// TIA Portal V17 export
// export: Created 2023-10-18T08:31:00.1217102Z, ExportSetting WithDefaults, WithReadOnly, DisplayName Totally Integrated Automation Portal, DisplayVersion V16 Update 4, DisplayName TIA Portal Version Control Interface, DisplayVersion V16 Update 2, DisplayName TIA Portal Openness, DisplayVersion V16 Update 4, DisplayName SINAMICS Startdrive Advanced, DisplayVersion V16 Update 5, DisplayName SINAMICS Startdrive G130, G150, S120, S150, SINAMICS MV, S210, DisplayVersion V16 Update 5, DisplayName SINAMICS Startdrive G110M, G120, G120C, G120D, G120P, G115D, DisplayVersion V16 Update 5, DisplayName STEP 7 Professional, DisplayVersion V16 Update 4, DisplayName STEP 7 Safety, DisplayVersion V16, DisplayName SINUMERIK 840D sl STEP 7 Toolbox, DisplayVersion V16 Update 2, DisplayName WinCC Advanced, DisplayVersion V16 Update 4
FUNCTION "AF_Safety" : Void   // FC2, FBD
{ S7_Optimized_Access := 'TRUE' }
VERSION : 0.1
// stored: AutoNumber true, CodeModifiedDate 2023-08-03T13:12:21.5628456Z, CompileDate 2023-08-03T13:12:26.4065718Z, CreationDate 2023-06-02T14:39:29.8490668Z, HandleErrorsWithinBlock false, InterfaceModifiedDate 2023-06-02T14:39:29.8490668Z, IsConsistent true, IsIECCheckEnabled false, IsKnowHowProtected false, IsWriteProtected false, LibraryConformanceStatus Error: The block contains calls of single instances. Warning: The object contains access to global data blocks. Warning: The block contains direct access to inputs, outputs, bit memories, indirect access to the registry or indirect access to external memory areas that are unknown at the time of compilation., ModifiedDate 2023-08-03T13:12:21.5628456Z, ParameterModified 2023-06-02T14:39:29.8490668Z, PLCSimAdvancedSupport true, SetENOAutomatically false, StructureModified 2023-06-02T14:39:29.8490668Z, UDAEnableTagReadback false
BEGIN

REGION Network 1
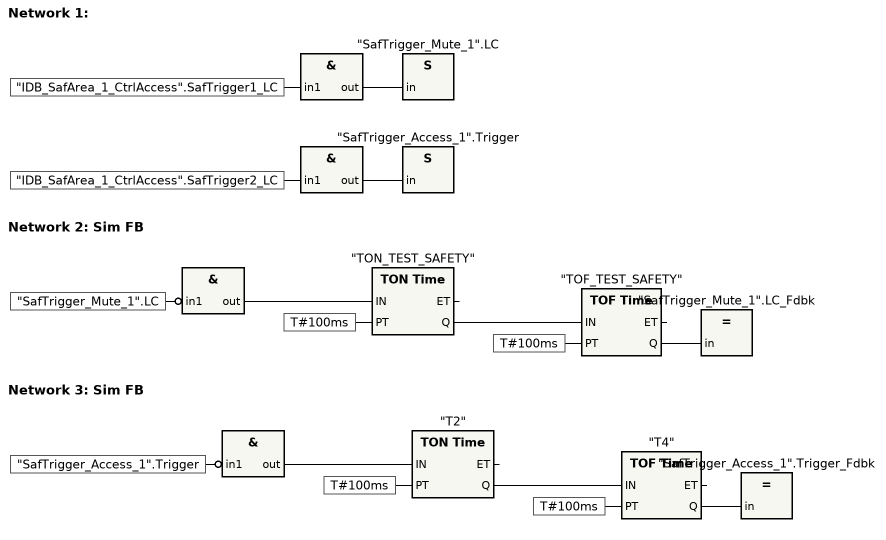
   IF "IDB_SafArea_1_CtrlAccess".SafTrigger1_LC THEN "SafTrigger_Mute_1".LC := TRUE; END_IF;
   IF "IDB_SafArea_1_CtrlAccess".SafTrigger2_LC THEN "SafTrigger_Access_1".Trigger := TRUE; END_IF;
END_REGION

REGION Network 2: Sim FB
   "TON_TEST_SAFETY".TON(IN := NOT "SafTrigger_Mute_1".LC, PT := T#100ms);
   "TOF_TEST_SAFETY".TOF(IN := "TON_TEST_SAFETY".Q, PT := T#100ms);
   "SafTrigger_Mute_1".LC_Fdbk := "TOF_TEST_SAFETY".Q;
END_REGION

REGION Network 3: Sim FB
   "T2".TON(IN := NOT "SafTrigger_Access_1".Trigger, PT := T#100ms);
   "T4".TOF(IN := "T2".Q, PT := T#100ms);
   "SafTrigger_Access_1".Trigger_Fdbk := "T4".Q;
END_REGION
END_FUNCTION
